FUNCTION TryConvert_DATE_TO_STRING : BOOL
VAR_INPUT
	in : DATE;
	out : REFERENCE TO STRING;
END_VAR

out := DATE_TO_STRING(in);
TryConvert_DATE_TO_STRING := TRUE;

END_FUNCTION

(* stored: Version 1.1.0.1, ProductVersion 3.1.4024.12
   POU TryConvert_DATE_TO_STRING: Id {2f428699-cb36-4d2e-a805-48822ba93951}, SpecialFunc None *)
